// TwinCAT 3 PLC project PLC1
// ProgramVersion: 3.1.4023.0
// libraries:
//   Tc2_SerialCom, * (Beckhoff Automation GmbH)
//   Tc2_Standard, * (Beckhoff Automation GmbH)
//   Tc2_System, * (Beckhoff Automation GmbH)
//   Tc3_Module, * (Beckhoff Automation GmbH)
// project tree:
//   DUTs/ ST_DeviceCount.TcDUT
//   / FastTask.TcTTO, PlcTask.TcTTO
//   GVLs/ GVL.TcGVL
//   POUs/ MAIN.TcPOU
// real-time tasks:
//   TASK PlcTask: cycle T#10ms, priority 20, ADS port 350
//   TASK FastTask: cycle T#2ms, priority 1, ADS port 351

CONFIGURATION PLC1
    RESOURCE PLC ON TwinCAT3
        TASK FastTask(INTERVAL := T#2ms, PRIORITY := 1);
        TASK PlcTask(INTERVAL := T#10ms, PRIORITY := 20);
        PROGRAM MAIN WITH PlcTask : MAIN;
    END_RESOURCE
END_CONFIGURATION

// ---- DUTs/ST_DeviceCount.TcDUT
TYPE ST_DeviceCount:
STRUCT
	aId: ARRAY[1..4] OF BYTE;
	nCount: DINT := 0;
END_STRUCT
END_TYPE

// ---- GVLs/GVL.TcGVL
{attribute 'qualified_only'}
VAR_GLOBAL
	TxBuffer: ComBuffer;
	RxBuffer: ComBuffer;
END_VAR

// ---- POUs/MAIN.TcPOU
PROGRAM MAIN
VAR
	i: INT;
	
	nState: INT;
	aReceiveData: ARRAY[1..4] OF BYTE;
	sDeviceId: STRING(80);
	
	nCursor: INT := 1;
	nRegconizedDeviceIds: INT;
	nTotalDevices: INT;
	aNullId: ARRAY[1..4] OF BYTE;
	aDeviceCount: ARRAY[1..10] OF ST_DeviceCount;
	bAddNewId: BOOL;
	fbRTrigAddNewId: R_TRIG;
END_VAR

CASE nState OF
	0: // Check if any data is received
		fbRTrigAddNewId(CLK:= bAddNewId, Q=> );
		IF fbRTrigAddNewId.Q AND (aReceiveData[1] <> 0) AND (aReceiveData[2] <> 0) AND (aReceiveData[3] <> 0) AND (aReceiveData[4] <> 0) THEN
			nState := nState + 1;
		END_IF
	1: // Get the barcode and check whether it was regconized
		sDeviceId := '';
		FOR i := 1 TO 4 DO
			sDeviceId := CONCAT(sDeviceId, CHR(aReceiveData[i]));
		END_FOR
		nState := 2;		
		FOR i := 1 TO 10 DO
			IF MEMCMP(ADR(aDeviceCount[i].aId), ADR(aReceiveData), 4) = 0 THEN
				nState := 3;
				EXIT;
			END_IF
		END_FOR
	2: // Realize the received barcode as a new barcode which was not known before
		IF nCursor < 11 THEN
			MEMCPY(ADR(aDeviceCount[nCursor].aId), ADR(aReceiveData), 4);
			nRegconizedDeviceIds := nRegconizedDeviceIds + 1;
			nCursor := nCursor + 1;
			nState := nState + 1;
		ELSE
			nState := 100;		
		END_IF
	3: // Increase the number of time the received bar code read
		FOR i := 1 TO 10 DO
			IF MEMCMP(ADR(aDeviceCount[i].aId), ADR(aReceiveData), 4) = 0 THEN
				aDeviceCount[i].nCount := aDeviceCount[i].nCount + 1;
				EXIT;
			END_IF
		END_FOR
		nTotalDevices := nTotalDevices + 1;
		nState := 0;
END_CASE

END_PROGRAM
